ADAPTER ECBusAdapter (* EtherCAT bus adapter between master, devices, and modules *)
  (* Standard: 61499-1; Description: Copyright (c) 2026 Sichuan Qunyuan Technology Co., Ltd. This program and the accompanying materials are made available under the terms of the Eclipse Public License 2.0 which is available at https://www.eclipse.org/legal/epl-2.0/ SPDX-License-Identifier: EPL-2.0 *)
  (* Version 1.0, 2026-04-09, Zijun Tang *)
  PACKAGE eclipse4diac::io::ethercat;
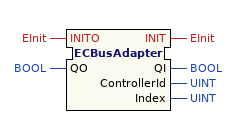
  EVENT_INPUT
    INITO : EInit; (* Initialization Confirm *)
  END_EVENT
  EVENT_OUTPUT
    INIT : EInit; (* Service Initialization *)
  END_EVENT
  VAR_INPUT
    QO : BOOL;
  END_VAR
  VAR_OUTPUT
    QI : BOOL;
    ControllerId : UINT;
    Index : UINT;
  END_VAR
END_ADAPTER
